// TIA Portal V20 export
DATA_BLOCK "HmiInterface"   // DB131
// stored: Access Published, MemoryReserve 100, Namespace Unit1.Em13
   VAR
      em : "LAF_typeEmInterface";
      cm : "Unit1.Em13.typeCmHmiInterface";
      jrUnloadingPnP : "LER_typeSequenceInterface";
      cmJRUnloadingPnPSafetyPin : "LBC_typeDigitalSignalInterface";
      cmJRUnloadingPnPJRDetect : "LBC_typeDigitalSignalInterface";
   END_VAR
   VAR RETAIN
      cmJRUnloadingPnPAxisX : "LBC_typeAxis64PosInterface";
      cmJRUnloadingPnPAxisZ : "LBC_typeAxis64PosInterface";
      cmJRUnloadingPnPAxisC : "LBC_typeAxis64PosInterface";
   END_VAR
   VAR
      cmJRUnloadingPnPClampOpenClose : "LBC_typeTwoWayActuatorInterface";
      intCondition : "Unit1.Em13.typeIntConditionHmiInterface";
   END_VAR
BEGIN
END_DATA_BLOCK
